# EPICS substitutions: siteApps-725b29e158e8061764313f5708af9e46fe30c0a8/siteApps-725b29e158e8061764313f5708af9e46fe30c0a8/Tr3/tr3App/Db/userHost.substitutions
# Example substitutions file

file "db/dbExample1.db" {
    { user = "sileeHost" }
}

file db/dbExample2.db {
    pattern { user, no, scan }
        { "sileeHost", 1, "1 second" }
        { "sileeHost", 2, "2 second" }
        { "sileeHost", 3, "5 second" }
}
